// TIA Portal V20 export
TYPE "s_zc_MiscInterlocks"
// stored: Access Published, IsFailsafeCompliant true, Namespace Safety
   STRUCT
      Misc_Int1 : Int;
      Misc_Int2 : Int;
      Misc_Int3 : Int;
      Misc_Int4 : Int;
      Misc_Int5 : Int;
      Misc_Int6 : Int;
      Misc_Int7 : Int;
      Misc_Int8 : Int;
      Misc_Int9 : Int;
      Misc_DInt1 : DInt;
      Misc_DInt2 : DInt;
      Misc_DInt3 : DInt;
      Misc_DInt4 : DInt;
      Misc_DInt5 : DInt;
   END_STRUCT;
END_TYPE
